// TIA Portal V21 export
FUNCTION "FaceplateFc" : Void   // FC102, LAD
{ S7_Optimized_Access := 'TRUE' }
// stored: AutoNumber false, SetENOAutomatically false
BEGIN

REGION Network 1 (SCL): Valve Open
   "ValveManualMode".Cv01 := "DO_FaceplateDb".Cv01.ValveOpen;
   "ValveManualMode".Cv01 := "DO_FaceplateDb".Cv01.ValveOpen;
   "ValveManualMode".Cv02 := "DO_FaceplateDb".Cv02.ValveOpen;
   "ValveManualMode".Cv03 := "DO_FaceplateDb".Cv03.ValveOpen;
   "ValveManualMode".Cv04 := "DO_FaceplateDb".Cv04.ValveOpen;
   "ValveManualMode".Cv05 := "DO_FaceplateDb".Cv05.ValveOpen;
   "ValveManualMode".Cv06 := "DO_FaceplateDb".Cv06.ValveOpen;
   "ValveManualMode".Cv07 := "DO_FaceplateDb".Cv07.ValveOpen;
   "ValveManualMode".Cv08 := "DO_FaceplateDb".Cv08.ValveOpen;
   "ValveManualMode".Cv09 := "DO_FaceplateDb".Cv09.ValveOpen;
   "ValveManualMode".Cv10 := "DO_FaceplateDb".Cv10.ValveOpen;
   "ValveManualMode".Cv11 := "DO_FaceplateDb".Cv11.ValveOpen;
   "ValveManualMode".Cv12 := "DO_FaceplateDb".Cv12.ValveOpen;
   "ValveManualMode".Cv13 := "DO_FaceplateDb".Cv13.ValveOpen;
   "ValveManualMode".Cv14 := "DO_FaceplateDb".Cv14.ValveOpen;
   "ValveManualMode".Cv15 := "DO_FaceplateDb".Cv15.ValveOpen;
   "ValveManualMode".Cv16 := "DO_FaceplateDb".Cv16.ValveOpen;
   "ValveManualMode".Cv17 := "DO_FaceplateDb".Cv17.ValveOpen;
   "ValveManualMode".Cv18 := "DO_FaceplateDb".Cv18.ValveOpen;
   "ValveManualMode".Cv19 := "DO_FaceplateDb".Cv19.ValveOpen;
   "ValveManualMode".Cv20 := "DO_FaceplateDb".Cv20.ValveOpen;
   "ValveManualMode".Cv21 := "DO_FaceplateDb".Cv21.ValveOpen;
   "ValveManualMode".Cv22 := "DO_FaceplateDb".Cv22.ValveOpen;
   "ValveManualMode".Cv23 := "DO_FaceplateDb".Cv23.ValveOpen;
   "ValveManualMode".Cv24 := "DO_FaceplateDb".Cv24.ValveOpen;
   "ValveManualMode".Cv25 := "DO_FaceplateDb".Cv25.ValveOpen;
   "ValveManualMode".Cv26 := "DO_FaceplateDb".Cv26.ValveOpen;
   "ValveManualMode".Cv27 := "DO_FaceplateDb".Cv27.ValveOpen;
   "ValveManualMode".Cv28 := "DO_FaceplateDb".Cv28.ValveOpen;
   "ValveManualMode".Cv29 := "DO_FaceplateDb".Cv29.ValveOpen;
   "ValveManualMode".Cv30 := "DO_FaceplateDb".Cv30.ValveOpen;
   "ValveManualMode".Cv31 := "DO_FaceplateDb".Cv31.ValveOpen;
   "ValveManualMode".Cv32 := "DO_FaceplateDb".Cv32.ValveOpen;
   "ValveManualMode".Cv33 := "DO_FaceplateDb".Cv33.ValveOpen;
   "ValveManualMode".Cv34 := "DO_FaceplateDb".Cv34.ValveOpen;
   "ValveManualMode".Cv35 := "DO_FaceplateDb".Cv35.ValveOpen;
   "ValveManualMode".Cv36 := "DO_FaceplateDb".Cv36.ValveOpen;
   "ValveManualMode".Cv37 := "DO_FaceplateDb".Cv37.ValveOpen;
   "ValveManualMode".Cv38 := "DO_FaceplateDb".Cv38.ValveOpen;
   "ValveManualMode".Cv39 := "DO_FaceplateDb".Cv39.ValveOpen;
   "ValveManualMode".Cv40 := "DO_FaceplateDb".Cv40.ValveOpen;
   "ValveManualMode".Cv41 := "DO_FaceplateDb".Cv41.ValveOpen;
   "ValveManualMode".Cv42 := "DO_FaceplateDb".Cv42.ValveOpen;
   "ValveManualMode".Cv43 := "DO_FaceplateDb".Cv43.ValveOpen;
   "ValveManualMode".Cv44 := "DO_FaceplateDb".Cv44.ValveOpen;
   "ValveManualMode".Cv45 := "DO_FaceplateDb".Cv45.ValveOpen;
   "ValveManualMode".Cv46 := "DO_FaceplateDb".Cv46.ValveOpen;
   "ValveManualMode".Cv47 := "DO_FaceplateDb".Cv47.ValveOpen;
   "ValveManualMode".Cv48 := "DO_FaceplateDb".Cv48.ValveOpen;
   "ValveManualMode".Cv49 := "DO_FaceplateDb".Cv49.ValveOpen;
   "ValveManualMode".Cv50 := "DO_FaceplateDb".Cv50.ValveOpen;
   "ValveManualMode".Cv51 := "DO_FaceplateDb".Cv51.ValveOpen;
   "ValveManualMode".Cv52 := "DO_FaceplateDb".Cv52.ValveOpen;
   "ValveManualMode".Cv53 := "DO_FaceplateDb".Cv53.ValveOpen;
   "ValveManualMode".Cv54 := "DO_FaceplateDb".Cv54.ValveOpen;
   "ValveManualMode".Cv55 := "DO_FaceplateDb".Cv55.ValveOpen;
   "ValveManualMode".Cv56 := "DO_FaceplateDb".Cv56.ValveOpen;
   "ValveManualMode".Cv57 := "DO_FaceplateDb".Cv57.ValveOpen;
   "ValveManualMode".Cv58 := "DO_FaceplateDb".Cv58.ValveOpen;
   "ValveManualMode".Cv59 := "DO_FaceplateDb".Cv59.ValveOpen;
   "ValveManualMode".Cv60 := "DO_FaceplateDb".Cv60.ValveOpen;
   "ValveManualMode".Cv61 := "DO_FaceplateDb".Cv61.ValveOpen;
   "ValveManualMode".Cv62 := "DO_FaceplateDb".Cv62.ValveOpen;
   "ValveManualMode".Cv63 := "DO_FaceplateDb".Cv63.ValveOpen;
   "ValveManualMode".Cv64 := "DO_FaceplateDb".Cv64.ValveOpen;
   "ValveManualMode".Fbov01 := "DO_FaceplateDb".Fbov01.ValveOpen;
END_REGION

REGION Network 2 (SCL): Pump Command
   "DoManualModeDb".Mm01Cmd :="DO_FaceplateDb"."Mm01 Ref".ValveOpen;
   "DoManualModeDb".Cp01Cmd := "DO_FaceplateDb"."Cp01 Ref".ValveOpen;


   //"DoDb".Do01.OpenClose := "DO_FaceplateDb"."Mm01 Ref".ValveOpen;
   //"DoDb".Do02.OpenClose := "DO_FaceplateDb"."Cp01 Ref".ValveOpen;
END_REGION

REGION Network 3 (SCL): Analog Output
   //Actual Rpm

   "Ao_Faceplate_Db".Mm01Ref.ActualRpm := "AoDb".Ao01.ActualRpm;
   "Ao_Faceplate_Db".Cp01Ref.ActualRpm:= "AoDb".Ao02.ActualRpm;


   //Min. Opeating Rpm
   // "AoDb".Ao01.MinOperatingRpm := "Ao_Faceplate_Db".CP01.MinOperating;
   //"AoDb".Ao02.MinOperatingRpm := "Ao_Faceplate_Db".MM01.MinOperating;
   "Ao_Faceplate_Db".Mm01Ref.MinOperating:= "AoDb".Ao01.MinOperatingRpm;
   "Ao_Faceplate_Db".Cp01Ref.MinOperating := "AoDb".Ao02.MinOperatingRpm;

   //Max. Operating Rpm
   "Ao_Faceplate_Db".Mm01Ref.MaxOperating:=  "AoDb".Ao01.MaxOperatingRpm;
   "Ao_Faceplate_Db".Cp01Ref.MaxOperating:= "AoDb".Ao02.MaxOperatingRpm;

   //Maximum Rpm
   // "AoDb".Ao01.MaxRpm := "Ao_Faceplate_Db".CP01.Maximum;
   // "AoDb".Ao02.MaxRpm := "Ao_Faceplate_Db".MM01.Maximum;
   "Ao_Faceplate_Db".Mm01Ref.Maximum:= "AoDb".Ao01.MaxRpm;
   "Ao_Faceplate_Db".Cp01Ref.Maximum:= "AoDb".Ao02.MaxRpm;

   //Manual Rpm
   // "AoDb".Ao01.ManualRpm := "Ao_Faceplate_Db".CP01.Manual;
   // "AoDb".Ao02.ManualRpm := "Ao_Faceplate_Db".MM01.Manual;
   "Ao_Faceplate_Db".Mm01Ref.Manual := "AoDb".Ao01.ManualRpm;
   "Ao_Faceplate_Db".Cp01Ref.Manual:= "AoDb".Ao02.ManualRpm;
END_REGION

REGION Network 4 (SCL): Analog Input
   // Moving Int value for units, 0 - Degree Celcius, 1 - bar, 2 - 

   // //"Ai_Faceplate_Db".Ai01.Unit := 0; spare
   // //"Ai_Faceplate_Db".Ai02.Unit := 0; spare
   // "Ai_Faceplate_Db".Ai03.Unit := 0;
   // "Ai_Faceplate_Db".Ai04.Unit := 0;
   // "Ai_Faceplate_Db".Ai05.Unit := 0;
   // "Ai_Faceplate_Db".Ai06.Unit := 0;
   // "Ai_Faceplate_Db".Ai07.Unit := 0;
   // "Ai_Faceplate_Db".Ai08.Unit := 1;
   // "Ai_Faceplate_Db".Ai09.Unit := 2;
   // "Ai_Faceplate_Db".Ai10.Unit := 3;
   // "Ai_Faceplate_Db".Ai11.Unit := 4;
END_REGION

REGION Network 5 (SCL)
   // "ValveDb".Cv01.OpenClose := "DO_FaceplateDb".Cv01.ValveOpen;
END_REGION
END_FUNCTION
